(* PLC project ST_IF_AND_ASSIGNMENT_1, Beckhoff Automation GmbH TwinCAT PLC Control 3.5.10.30 *)
(* stored: creationDateTime 2019-09-26T11:42:34.782397, modificationDateTime 2019-09-26T11:42:34.7853953 *)

PROGRAM MAIN
VAR

	Present: INT;
	Open: INT;
	Close: INT;
	Workpiece: BOOL;
	SENSOR: BOOL;
	Gate: INT;
END_VAR

                  
Gate := Close;
IF (SENSOR AND Workpiece) THEN
     Gate := Open;
    ELSE
     Gate := Close;
END_IF;


                
END_PROGRAM

CONFIGURATION Application
  RESOURCE ST_Evolution_1 ON PLC
    TASK PlcTask(INTERVAL := T#0ms, PRIORITY := 20);
    PROGRAM MAIN WITH PlcTask : MAIN;
  END_RESOURCE
END_CONFIGURATION
